// TIA Portal V17 export
// export: Created 2024-09-03T21:54:54.0406379Z, ExportSetting WithDefaults, DisplayName Totally Integrated Automation Portal, DisplayVersion V17 Update 7, DisplayName TIA Portal Openness, DisplayVersion V17 Update 7, DisplayName TIA Portal Version Control Interface, DisplayVersion V17, DisplayName SINAMICS Startdrive Advanced, DisplayVersion V17 SP2, DisplayName SINAMICS Startdrive G110M, G120, G120C, G120D, G120P, G115D, DisplayVersion V17 SP2, DisplayName SINAMICS Startdrive G130, G150, S120, S150, SINAMICS MV, S210, DisplayVersion V17 SP2, DisplayName STEP 7 Professional, DisplayVersion V17 Update 7, DisplayName STEP 7 Safety, DisplayVersion V17 Update 6, DisplayName WinCC Advanced / Unified PC, DisplayVersion V17 Update 7
FUNCTION_BLOCK "FB_Main"   // FB5000, LAD
{ S7_Optimized_Access := 'TRUE' }
VERSION : 0.1
// stored: AutoNumber false, IsIECCheckEnabled false, IsRetainMemResEnabled false, MemoryReserve 100, SetENOAutomatically false, UDAEnableTagReadback false
   VAR
      IEC_Timer_0_Instance { S7_SetPoint := 'True'} : TON_TIME;
      MachineModeOld { S7_SetPoint := 'True'} : UInt;
      F_TRIG_Instance { S7_SetPoint := 'True'} : F_TRIG;
      F_TRIG_Instance_1 { S7_SetPoint := 'True'} : F_TRIG;
      F_TRIG_Instance_2 { S7_SetPoint := 'True'} : F_TRIG;
      R_TRIG_Instance { S7_SetPoint := 'True'} : R_TRIG;
      R_TRIG_Instance_1 { S7_SetPoint := 'True'} : R_TRIG;
   END_VAR
   VAR_TEMP   // added for the SCL form of the ladder/FBD networks
      _w1 : Bool;
      _w2 : Bool;
   END_VAR
BEGIN

REGION Network 1: alarms fc, lamp fc
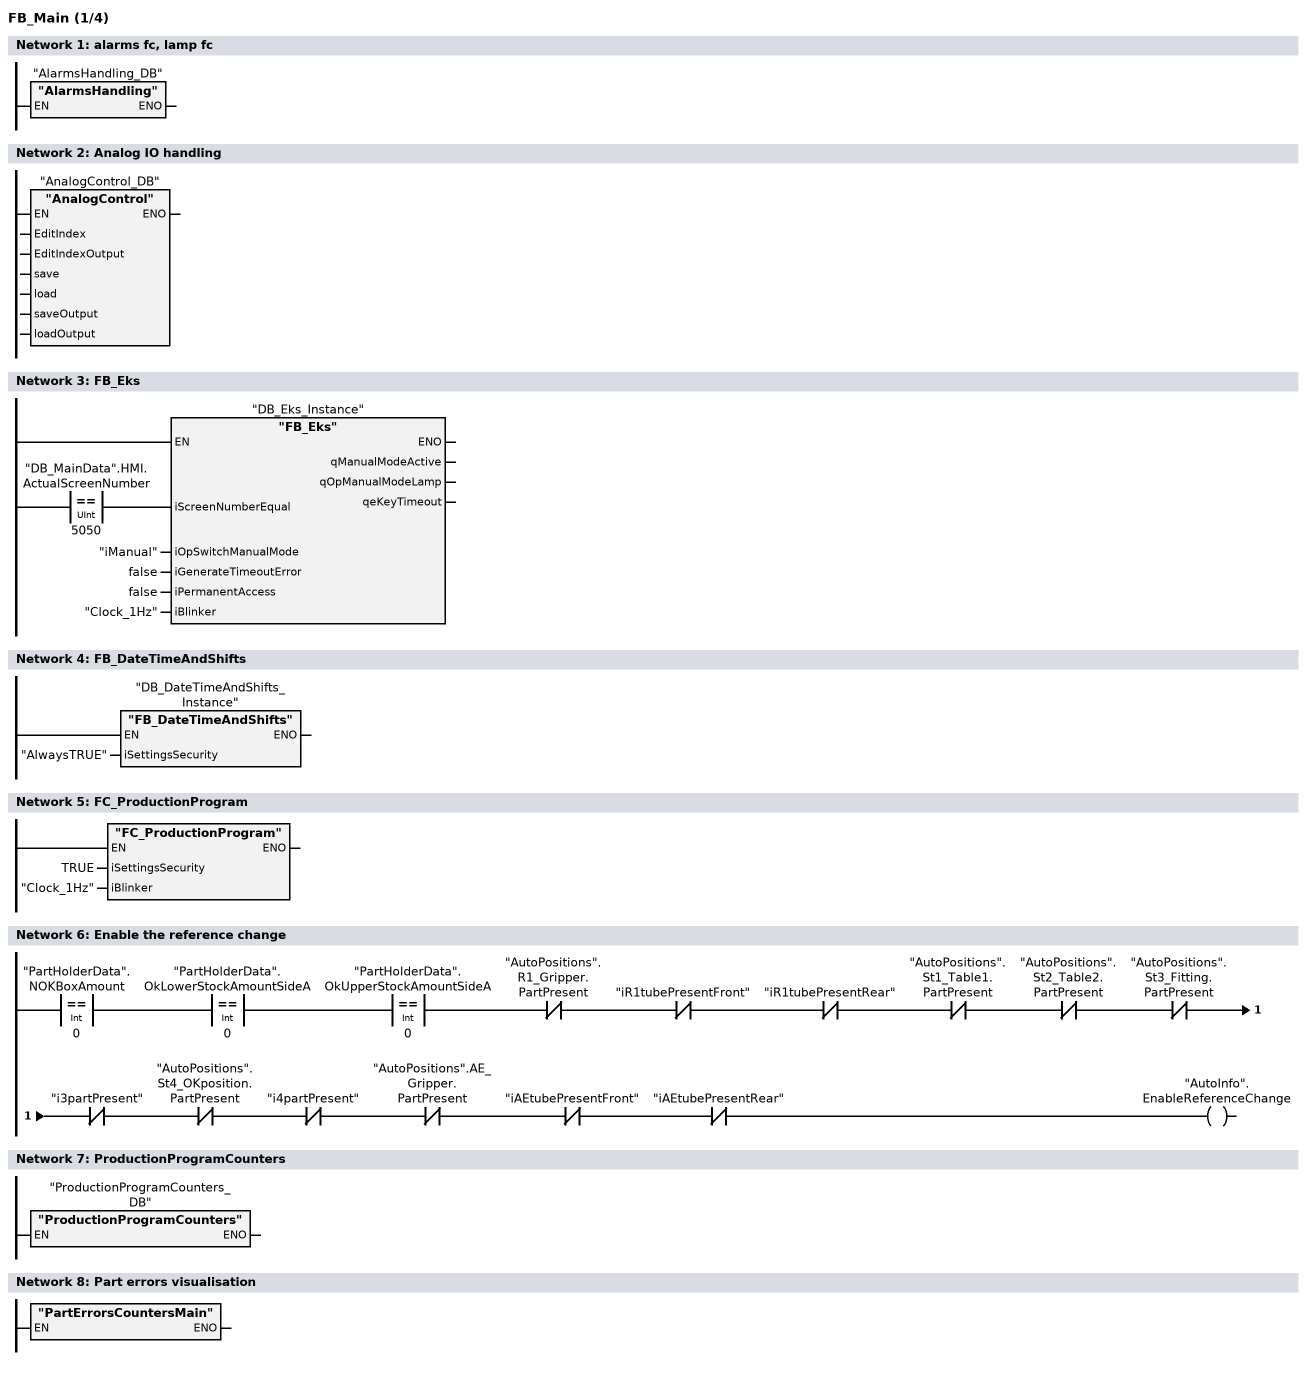
   RUNG wire#powerrail
      "AlarmsHandling_DB"()
   END_RUNG
   // the same network as SCL:
   "AlarmsHandling_DB"();   // "AlarmsHandling"
END_REGION

REGION Network 2: Analog IO handling
   RUNG wire#powerrail
      "AnalogControl_DB"(EditIndex :=, save :=, load :=, EditIndexOutput :=, saveOutput :=, loadOutput :=)
   END_RUNG
   // the same network as SCL:
   "AnalogControl_DB"();   // "AnalogControl"
END_REGION

REGION Network 3: FB_Eks
   RUNG wire#powerrail
      "DB_Eks_Instance"(iScreenNumberEqual := wire#w1, iOpSwitchManualMode := "iManual", iGenerateTimeoutError := false, iPermanentAccess := false, iBlinker := "Clock_1Hz", qManualModeActive =>, qOpManualModeLamp =>, qeKeyTimeout =>)
   END_RUNG
   RUNG wire#powerrail
      { S7_Templates := "SrcType := UInt" } EQ_Contact(in1 := "DB_MainData".HMI.ActualScreenNumber, in2 := 5050)
   END_RUNG wire#w1
   // the same network as SCL:
   "DB_Eks_Instance"(iScreenNumberEqual := "DB_MainData".HMI.ActualScreenNumber = 5050,   // "FB_Eks"
                     iOpSwitchManualMode := "iManual",
                     iGenerateTimeoutError := false,
                     iPermanentAccess := false,
                     iBlinker := "Clock_1Hz");
END_REGION

REGION Network 4: FB_DateTimeAndShifts
   RUNG wire#powerrail
      "DB_DateTimeAndShifts_Instance"(iSettingsSecurity := "AlwaysTRUE")
   END_RUNG
   // the same network as SCL:
   "DB_DateTimeAndShifts_Instance"(iSettingsSecurity := "AlwaysTRUE");   // "FB_DateTimeAndShifts"
END_REGION

REGION Network 5: FC_ProductionProgram
   RUNG wire#powerrail
      "FC_ProductionProgram"(iSettingsSecurity := TRUE, iBlinker := "Clock_1Hz")
   END_RUNG
   // the same network as SCL:
   "FC_ProductionProgram"(iSettingsSecurity := TRUE, iBlinker := "Clock_1Hz");
END_REGION

REGION Network 6: Enable the reference change
   RUNG wire#powerrail
      { S7_Templates := "SrcType := Int" } EQ_Contact(in1 := "PartHolderData".NOKBoxAmount, in2 := 0)
      { S7_Templates := "SrcType := Int" } EQ_Contact(in1 := "PartHolderData".OkLowerStockAmountSideA, in2 := 0)
      { S7_Templates := "SrcType := Int" } EQ_Contact(in1 := "PartHolderData".OkUpperStockAmountSideA, in2 := 0)
      I_Contact( "AutoPositions".R1_Gripper.PartPresent )
      I_Contact( "iR1tubePresentFront" )
      I_Contact( "iR1tubePresentRear" )
      I_Contact( "AutoPositions".St1_Table1.PartPresent )
      I_Contact( "AutoPositions".St2_Table2.PartPresent )
      I_Contact( "AutoPositions".St3_Fitting.PartPresent )
      I_Contact( "i3partPresent" )
      I_Contact( "AutoPositions".St4_OKposition.PartPresent )
      I_Contact( "i4partPresent" )
      I_Contact( "AutoPositions".AE_Gripper.PartPresent )
      I_Contact( "iAEtubePresentFront" )
      I_Contact( "iAEtubePresentRear" )
      Coil( "AutoInfo".EnableReferenceChange )
   END_RUNG
   // the same network as SCL:
   "AutoInfo".EnableReferenceChange := ("PartHolderData".NOKBoxAmount = 0) AND ("PartHolderData".OkLowerStockAmountSideA = 0) AND ("PartHolderData".OkUpperStockAmountSideA = 0) AND NOT "AutoPositions".R1_Gripper.PartPresent AND NOT "iR1tubePresentFront" AND NOT "iR1tubePresentRear" AND NOT "AutoPositions".St1_Table1.PartPresent AND NOT "AutoPositions".St2_Table2.PartPresent AND NOT "AutoPositions".St3_Fitting.PartPresent AND NOT "i3partPresent" AND NOT "AutoPositions".St4_OKposition.PartPresent AND NOT "i4partPresent" AND NOT "AutoPositions".AE_Gripper.PartPresent AND NOT "iAEtubePresentFront" AND NOT "iAEtubePresentRear";
END_REGION

REGION Network 7: ProductionProgramCounters
   RUNG wire#powerrail
      "ProductionProgramCounters_DB"()
   END_RUNG
   // the same network as SCL:
   "ProductionProgramCounters_DB"();   // "ProductionProgramCounters"
END_REGION

REGION Network 8: Part errors visualisation
   RUNG wire#powerrail
      "PartErrorsCountersMain"()
   END_RUNG
   // the same network as SCL:
   "PartErrorsCountersMain"();
END_REGION

REGION Network 9: FB_Devices
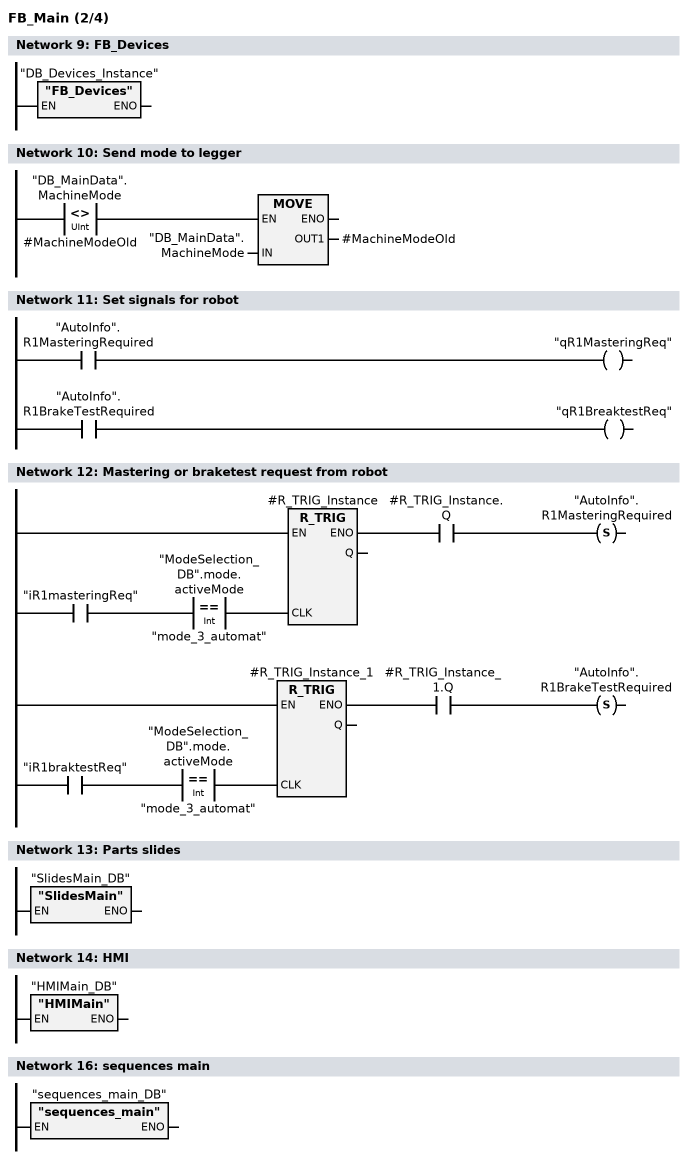
   RUNG wire#powerrail
      "DB_Devices_Instance"()
   END_RUNG
   // the same network as SCL:
   "DB_Devices_Instance"();   // "FB_Devices"
END_REGION

REGION Network 10: Send mode to legger
   RUNG wire#powerrail
      { S7_Templates := "SrcType := UInt" } NE_Contact(in1 := "DB_MainData".MachineMode, in2 := #MachineModeOld)
      Move(in := "DB_MainData".MachineMode, out1 => #MachineModeOld)
   END_RUNG
   // the same network as SCL:
   IF "DB_MainData".MachineMode <> #MachineModeOld THEN #MachineModeOld := "DB_MainData".MachineMode; END_IF;
END_REGION

REGION Network 11: Set signals for robot
   RUNG wire#powerrail
      Contact( "AutoInfo".R1MasteringRequired )
      Coil( "qR1MasteringReq" )
   END_RUNG
   RUNG wire#powerrail
      Contact( "AutoInfo".R1BrakeTestRequired )
      Coil( "qR1BreaktestReq" )
   END_RUNG
   // the same network as SCL:
   "qR1MasteringReq" := "AutoInfo".R1MasteringRequired;
   "qR1BreaktestReq" := "AutoInfo".R1BrakeTestRequired;
END_REGION

REGION Network 12: Mastering or braketest request from robot
   RUNG wire#powerrail
      #R_TRIG_Instance.R_TRIG(CLK := wire#w1, Q =>)
      Contact( #R_TRIG_Instance.Q )
      S_Coil( "AutoInfo".R1MasteringRequired )
   END_RUNG
   RUNG wire#powerrail
      Contact( "iR1masteringReq" )
      { S7_Templates := "SrcType := Int" } EQ_Contact(in1 := "ModeSelection_DB".mode.activeMode, in2 := "mode_3_automat")
   END_RUNG wire#w1
   RUNG wire#powerrail
      #R_TRIG_Instance_1.R_TRIG(CLK := wire#w2, Q =>)
      Contact( #R_TRIG_Instance_1.Q )
      S_Coil( "AutoInfo".R1BrakeTestRequired )
   END_RUNG
   RUNG wire#powerrail
      Contact( "iR1braktestReq" )
      { S7_Templates := "SrcType := Int" } EQ_Contact(in1 := "ModeSelection_DB".mode.activeMode, in2 := "mode_3_automat")
   END_RUNG wire#w2
   // the same network as SCL:
   #R_TRIG_Instance(CLK := "iR1masteringReq" AND ("ModeSelection_DB".mode.activeMode = "mode_3_automat"),   // R_TRIG
                    ENO => #_w1);
   IF #_w1 AND #R_TRIG_Instance.Q THEN "AutoInfo".R1MasteringRequired := TRUE; END_IF;
   #R_TRIG_Instance_1(CLK := "iR1braktestReq" AND ("ModeSelection_DB".mode.activeMode = "mode_3_automat"),   // R_TRIG
                      ENO => #_w2);
   IF #_w2 AND #R_TRIG_Instance_1.Q THEN "AutoInfo".R1BrakeTestRequired := TRUE; END_IF;
END_REGION

REGION Network 13: Parts slides
   RUNG wire#powerrail
      "SlidesMain_DB"()
   END_RUNG
   // the same network as SCL:
   "SlidesMain_DB"();   // "SlidesMain"
END_REGION

REGION Network 14: HMI
   RUNG wire#powerrail
      "HMIMain_DB"()
   END_RUNG
   // the same network as SCL:
   "HMIMain_DB"();   // "HMIMain"
END_REGION

REGION Network 15 (SCL): mode selection
   "ModeSelection_DB"(iSafetyOKauto := "safety_signals"."4L+" AND NOT "SandBoxData".resetAuto,
                      iSafetyOKmanual := "safety_signals"."3L+",
                      iBasePosition := "sq_carousel_main_".base AND "sq_carousel_main_"."Base done".X AND
                      "sq_carousel_insertion_st1".base AND "sq_carousel_insertion_st1"."Base done".X AND
                      "sq_carousel_unloading_st2".base AND "sq_carousel_unloading_st2"."Base done".X AND
                      "sq_fitting_station_st3".base AND "sq_fitting_station_st3"."Base done".X AND
                      "sq_autoeject_DB".base AND "sq_autoeject_DB"."Base done".X AND
   //                   "sq_hanger_manipulator".base AND "sq_hanger_manipulator"."Base done".X AND
                      "sq_robot_".base AND "sq_robot_"."Base done".X,
                      iBaseInManualMode := TRUE,
                      OFF_SQ := FALSE,
                      INIT_SQ := TRUE,
                      SW_AUTO := TRUE);

   "ModeSelection_DB".mode.switch.auto := "iAuto" AND NOT "iManual";
   "ModeSelection_DB".mode.button.basic.request.button := "iBtnBasicPosition";
   "ModeSelection_DB".mode.button.auto.startRequest.button := "iBtnStartAuto";

   "DB_MainData".MachineMode := INT_TO_UINT("ModeSelection_DB".mode.activeMode);
   "SystemHMI".ManualMode := "ModeSelection_DB".mode.activeMode = "mode_1_manual";
   "SystemHMI".GoToBasicPosition := "ModeSelection_DB".mode.activeMode = "mode_2_base";
   "SystemHMI".AutomaticMode := "ModeSelection_DB".mode.activeMode = "mode_3_automat" OR "ModeSelection_DB".mode.activeMode = "mode_4_semiautomat";
   "SystemHMI".ModeChanged := "ModeSelection_DB".mode.modeChanged;

   "qBasicPosition" :=
   "ModeSelection_DB"."Base position reached".X OR
   "ModeSelection_DB".mode.activeMode = "mode_2_base" AND "Clock_5Hz" OR
   "ModeSelection_DB".mode.button.basic.request.visibility AND "Clock_1Hz";

   "qAuto" :=
   "ModeSelection_DB".mode.activeMode = "mode_3_automat" OR
   "ModeSelection_DB".mode.activeMode = "mode_4_semiautomat" OR
   "ModeSelection_DB".mode.button.auto.startRequest.visibility AND "Clock_1Hz";

   "qManual" := "ModeSelection_DB".mode.activeMode = "mode_1_manual";
END_REGION

REGION Network 16: sequences main
   RUNG wire#powerrail
      "sequences_main_DB"()
   END_RUNG
   // the same network as SCL:
   "sequences_main_DB"();   // "sequences_main"
END_REGION

REGION Network 17
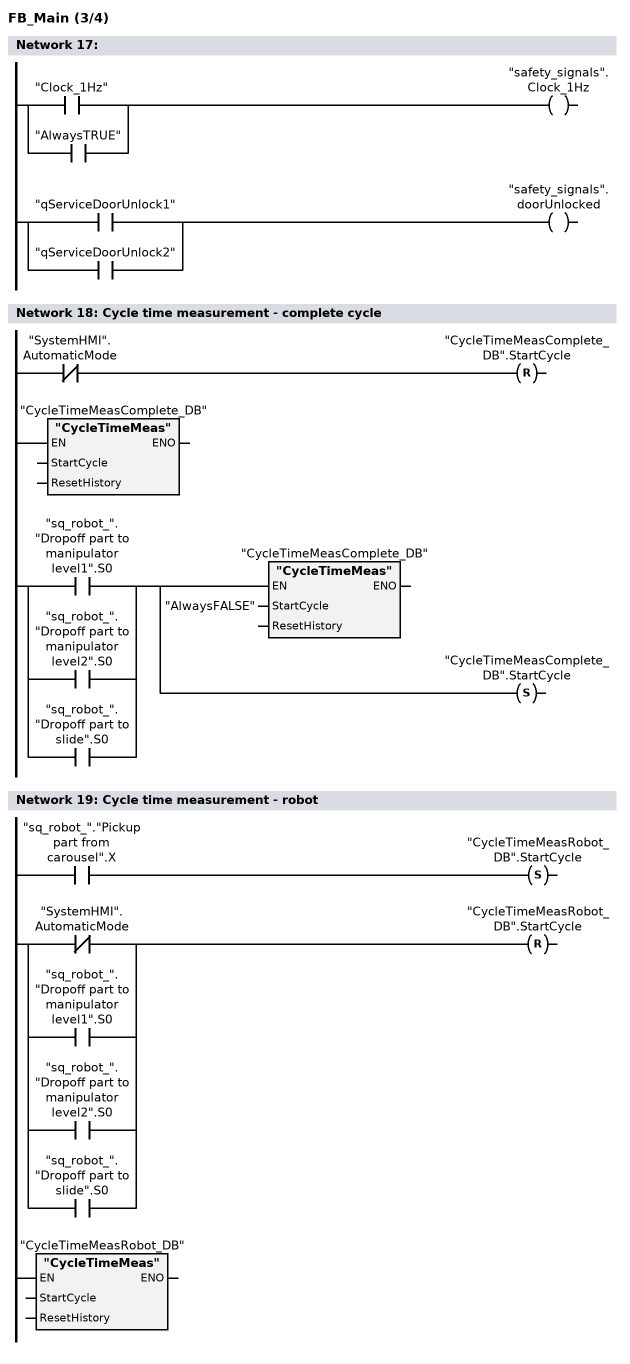
   RUNG wire#powerrail
      Contact( "Clock_1Hz" )
      wire#w1
      Coil( "safety_signals".Clock_1Hz )
   END_RUNG
   RUNG wire#powerrail
      Contact( "AlwaysTRUE" )
   END_RUNG wire#w1
   RUNG wire#powerrail
      Contact( "qServiceDoorUnlock1" )
      wire#w2
      Coil( "safety_signals".doorUnlocked )
   END_RUNG
   RUNG wire#powerrail
      Contact( "qServiceDoorUnlock2" )
   END_RUNG wire#w2
   // the same network as SCL:
   "safety_signals".Clock_1Hz := "Clock_1Hz" OR "AlwaysTRUE";
   "safety_signals".doorUnlocked := "qServiceDoorUnlock1" OR "qServiceDoorUnlock2";
END_REGION

REGION Network 18: Cycle time measurement - complete cycle
   RUNG wire#powerrail
      I_Contact( "SystemHMI".AutomaticMode )
      R_Coil( "CycleTimeMeasComplete_DB".StartCycle )
   END_RUNG
   RUNG wire#powerrail
      "CycleTimeMeasComplete_DB"(StartCycle :=, ResetHistory :=)
   END_RUNG
   RUNG wire#powerrail
      Contact( "sq_robot_"."Dropoff part to manipulator level1".S0 )
      wire#w1
      "CycleTimeMeasComplete_DB"(StartCycle := "AlwaysFALSE", ResetHistory :=)
   END_RUNG
   RUNG wire#powerrail
      Contact( "sq_robot_"."Dropoff part to manipulator level2".S0 )
   END_RUNG wire#w1
   RUNG wire#powerrail
      Contact( "sq_robot_"."Dropoff part to slide".S0 )
   END_RUNG wire#w1
   RUNG wire#w1
      S_Coil( "CycleTimeMeasComplete_DB".StartCycle )
   END_RUNG
   // the same network as SCL:
   IF NOT "SystemHMI".AutomaticMode THEN "CycleTimeMeasComplete_DB".StartCycle := FALSE; END_IF;
   "CycleTimeMeasComplete_DB"();   // "CycleTimeMeas"
   #_w1 := "sq_robot_"."Dropoff part to manipulator level1".S0 OR "sq_robot_"."Dropoff part to manipulator level2".S0 OR "sq_robot_"."Dropoff part to slide".S0;
   IF #_w1 THEN
       "CycleTimeMeasComplete_DB"(StartCycle := "AlwaysFALSE");   // "CycleTimeMeas"
       "CycleTimeMeasComplete_DB".StartCycle := TRUE;
   END_IF;
END_REGION

REGION Network 19: Cycle time measurement - robot
   RUNG wire#powerrail
      Contact( "sq_robot_"."Pickup part from carousel".X )
      S_Coil( "CycleTimeMeasRobot_DB".StartCycle )
   END_RUNG
   RUNG wire#powerrail
      I_Contact( "SystemHMI".AutomaticMode )
      wire#w1
      R_Coil( "CycleTimeMeasRobot_DB".StartCycle )
   END_RUNG
   RUNG wire#powerrail
      Contact( "sq_robot_"."Dropoff part to manipulator level1".S0 )
   END_RUNG wire#w1
   RUNG wire#powerrail
      Contact( "sq_robot_"."Dropoff part to manipulator level2".S0 )
   END_RUNG wire#w1
   RUNG wire#powerrail
      Contact( "sq_robot_"."Dropoff part to slide".S0 )
   END_RUNG wire#w1
   RUNG wire#powerrail
      "CycleTimeMeasRobot_DB"(StartCycle :=, ResetHistory :=)
   END_RUNG
   // the same network as SCL:
   IF "sq_robot_"."Pickup part from carousel".X THEN "CycleTimeMeasRobot_DB".StartCycle := TRUE; END_IF;
   IF NOT "SystemHMI".AutomaticMode OR "sq_robot_"."Dropoff part to manipulator level1".S0 OR "sq_robot_"."Dropoff part to manipulator level2".S0 OR "sq_robot_"."Dropoff part to slide".S0 THEN
       "CycleTimeMeasRobot_DB".StartCycle := FALSE;
   END_IF;
   "CycleTimeMeasRobot_DB"();   // "CycleTimeMeas"
END_REGION

REGION Network 20: Reset history
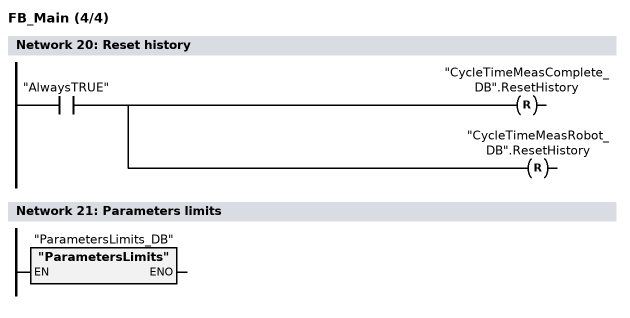
   RUNG wire#powerrail
      Contact( "AlwaysTRUE" )
      wire#w1
      R_Coil( "CycleTimeMeasComplete_DB".ResetHistory )
   END_RUNG
   RUNG wire#w1
      R_Coil( "CycleTimeMeasRobot_DB".ResetHistory )
   END_RUNG
   // the same network as SCL:
   IF "AlwaysTRUE" THEN
       "CycleTimeMeasComplete_DB".ResetHistory := FALSE;
       "CycleTimeMeasRobot_DB".ResetHistory := FALSE;
   END_IF;
END_REGION

REGION Network 21: Parameters limits
   RUNG wire#powerrail
      "ParametersLimits_DB"()
   END_RUNG
   // the same network as SCL:
   "ParametersLimits_DB"();   // "ParametersLimits"
END_REGION

REGION Network 22: Readings
END_REGION
END_FUNCTION_BLOCK
